# B&R Automation Studio project SFC
Automation Studio 4.12.2.93

## Configuration Config1

### Hardware
```
X20CP1584 : X20CP1584 v1.10.0.0
  Connector IF2:
    ActivateDevice = 1
  ConfigurationID = ExeBonusSFC_Config1
  Simulation = 1
  FileDevice1
  FileDeviceName1 = USER
  FileDevicePath1 = USER_PATH
```

## Logical view

### Program Logical/Program (IEC)

#### Cyclic.sfc - Cyclic code
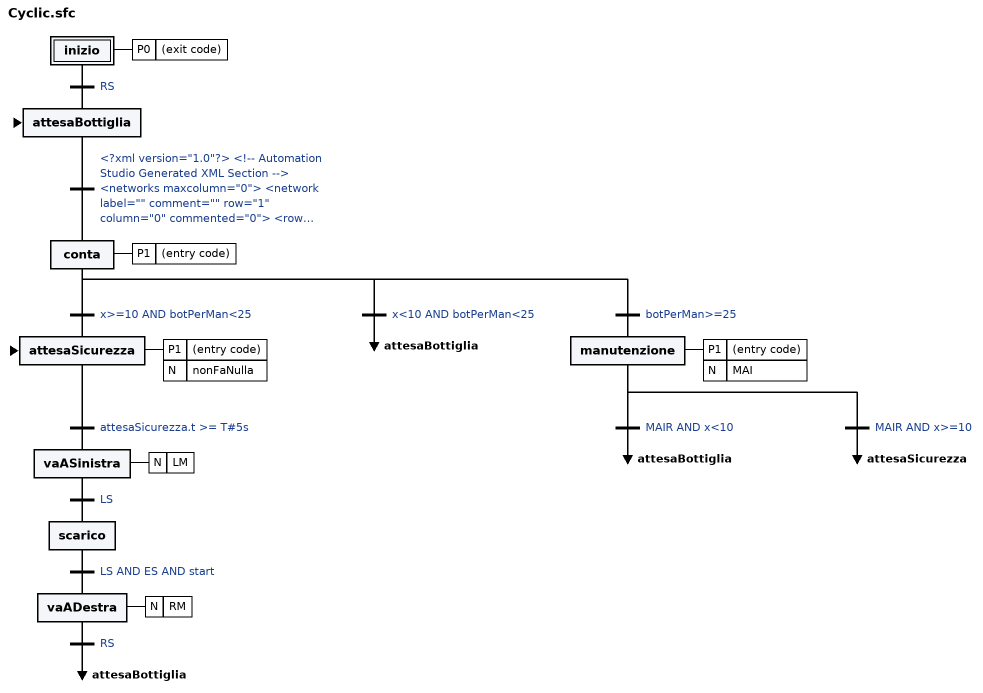
```iecst
PROGRAM _CYCLIC
INITIAL_STEP inizio:
END_STEP
EXIT_ACTION

(* Inizzializzazione delle variabili *)

x:= 0;
botPerMan:=0;
END_ACTION
TRANSITION FROM inizio TO attesaBottiglia:=
RS
END_TRANSITION
STEP attesaBottiglia:
END_STEP
TRANSITION fronte positivo fotocellula FROM attesaBottiglia TO conta:=
(* @LANGUAGE := 'ld' *)

<?xml version="1.0"?>
<!-- Automation Studio Generated XML Section -->
<networks maxcolumn="0">
	<network label="" comment="" row="1" column="0" commented="0">
		<row>
			<contact type="positive transition" name="CELL"/>
			<line/>
			<line/>
			<coil type="open" name="Transition"/>
		</row>
	</network>
</networks>

END_TRANSITION
STEP conta:
END_STEP
ENTRY_ACTION

(* TODO: Insert Program *)

x:=x+1;
CELL := FALSE;
botPerMan:=botPerMan+1;

END_ACTION
TRANSITION FROM conta TO attesaSicurezza:=
x>=10 AND botPerMan<25
END_TRANSITION
TRANSITION FROM conta TO attesaBottiglia:=
x<10 AND botPerMan<25
END_TRANSITION
(* @SFCISJUMP := 'attesaBottiglia' *)
TRANSITION FROM conta TO manutenzione:=
botPerMan>=25
END_TRANSITION
IEC_STEP manutenzione:
MAI(N);
END_STEP
ENTRY_ACTION

(* TODO: Insert Program *)

botPerMan:=0;
END_ACTION
TRANSITION FROM manutenzione TO attesaBottiglia:=
MAIR AND x<10
END_TRANSITION
(* @SFCISJUMP := 'attesaBottiglia' *)
TRANSITION FROM manutenzione TO attesaSicurezza:=
MAIR AND x>=10
END_TRANSITION
(* @SFCISJUMP := 'attesaSicurezza' *)
IEC_STEP attesaSicurezza:
nonFaNulla(N);
END_STEP
ENTRY_ACTION

(* TODO: Insert Program *)

x:=0;
END_ACTION
TRANSITION FROM attesaSicurezza TO vaASinistra:=
attesaSicurezza.t >= T#5s
END_TRANSITION
IEC_STEP vaASinistra:
LM(N);
END_STEP
TRANSITION FROM vaASinistra TO scarico:=
LS
END_TRANSITION
STEP scarico:
END_STEP
TRANSITION FROM scarico TO vaADestra:=
LS AND ES AND start
END_TRANSITION
IEC_STEP vaADestra:
RM(N);
END_STEP
TRANSITION FROM vaADestra TO attesaBottiglia:=
RS
END_TRANSITION
(* @SFCISJUMP := 'attesaBottiglia' *)
END_PROGRAM
```

#### Variables.var - Local variables
```iecst
VAR
	nonFaNulla : BOOL;
	botPerMan : USINT;
	x : USINT;
	RM : BOOL;
	LM : BOOL;
	MAI : BOOL;
	CELL : BOOL;
	LS : BOOL;
	RS : BOOL;
	ES : BOOL;
	start : BOOL;
	MAIR : BOOL;
END_VAR
```

Listed in the project but not available here: Logical/Program/Types.typ
